// TIA Portal V20 export
DATA_BLOCK "SP205"   // DB316
// stored: MemoryReserve 100
   VAR
      "MAIN OP PENDANT REQUIRED PL LAMP ON (YELLOW)" : Bool;
      SPARE : Bool;
      "MAIN OP HOME PBL LAMP ON (GREEN)" : Bool;
      SPARE_1 : Bool;
      SPARE_2 : Bool;
      SPARE_3 : Bool;
      SPARE_4 : Bool;
      "MAIN OP SCS MODE SELECT DISABLE PL LAMP ON (GREEN)" : Bool;
   END_VAR
BEGIN
END_DATA_BLOCK
